// TIA Portal V16 export
// export: Created 2021-07-03T21:22:42.5545027Z, ExportSetting WithDefaults, DisplayName Totally Integrated Automation Portal, DisplayVersion V16, DisplayName TIA Portal Version Control Interface, DisplayVersion V16, DisplayName TIA Portal Openness, DisplayVersion V16, DisplayName STEP 7 Professional, DisplayVersion V16, DisplayName STEP 7 Safety, DisplayVersion V16, DisplayName WinCC Professional, DisplayVersion V16
TYPE "118MK2_PlantIF_Status"
// stored: IsFailsafeCompliant false
   STRUCT
      PlantSeq_Data { S7_SetPoint := 'True'} : "PLANT_SEQ_STATE";
      Status_Data { S7_SetPoint := 'True'} : "118MK2_PlantData";   // Status Information from Machine
      Recipe_Data { S7_SetPoint := 'True'} : "118MK2_RecipeData";   // Recipe Information from Machine
   END_STRUCT;
END_TYPE
